FUNCTION WConcat5 : WSTRING(255)
VAR_INPUT
	wsExpression1: WSTRING(255);
	wsExpression2: WSTRING(255);
	wsExpression3: WSTRING(255);
	wsExpression4: WSTRING(255);
	wsExpression5: WSTRING(255);
END_VAR

WConcat5 := WCONCAT(wsExpression1, wsExpression2);
WConcat5 := WCONCAT(WConcat5, wsExpression3);
WConcat5 := WCONCAT(WConcat5, wsExpression4);
WConcat5 := WCONCAT(WConcat5, wsExpression5);

END_FUNCTION

(* stored: Version 1.1.0.1, ProductVersion 3.1.4024.11
   POU WConcat5: Id {53f4a1e3-33cc-4f4a-8ca4-cfb48f7e12ba}, SpecialFunc None *)
